// TIA Portal V19 export
FUNCTION_BLOCK "Area02_HU_FB"   // FB144, LAD
TITLE = AREA 01 HU PUMP
// stored: MemoryReserve 100, SetENOAutomatically false
   VAR_INPUT
      AreaInterface : "AreaInterface";
   END_VAR
   VAR_OUTPUT
      MachineInterface : "MachineInterface";
   END_VAR
   VAR
      Pump : "HU_Pump";
      Tank { S7_SetPoint := 'True'} : "HU_Tank";
      HMI : Struct
         Pressure_FinalCut : Real;
      END_STRUCT;
   END_VAR
   VAR_TEMP
      retval : Int;
      OilTemperature : Real;
      AnalTemperature_Real : Real;
      Delta : Real;
      Delta2 : Real;
   END_VAR
BEGIN

REGION Network 1: <<< PUMP >>>
END_REGION

REGION Network 2: Data In
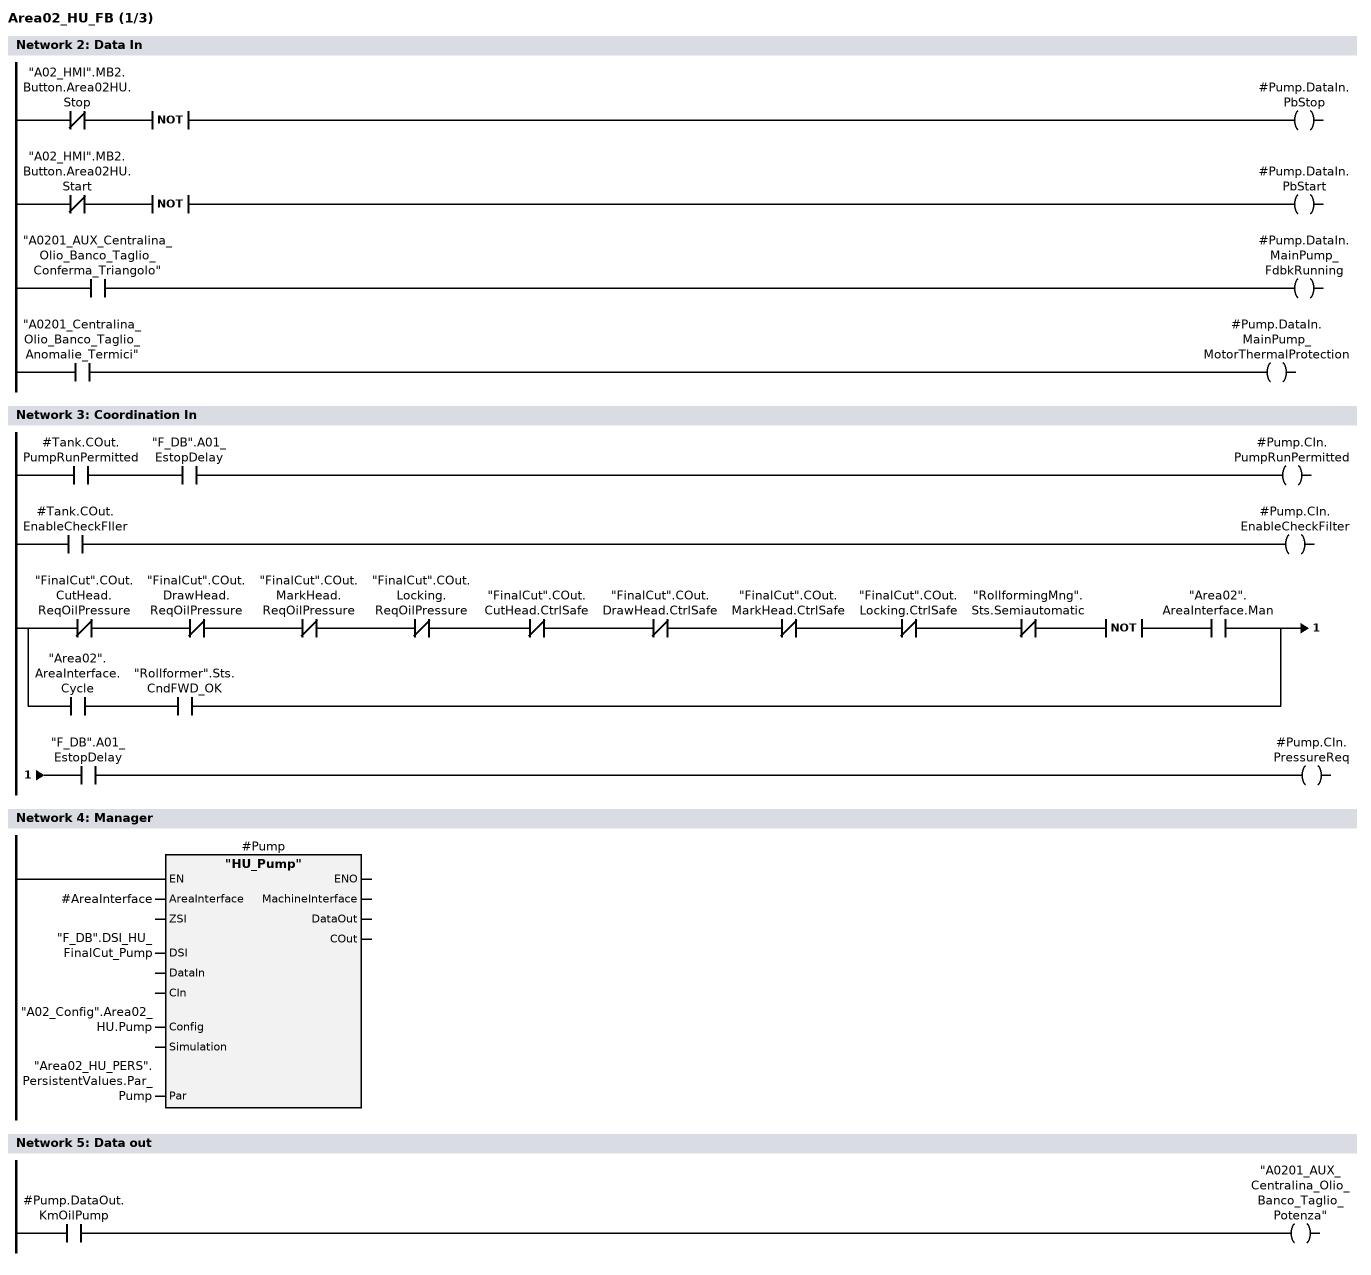
   RUNG wire#powerrail
      I_Contact( "A02_HMI".MB2.Button.Area02HU.Stop )
      Not()
      Coil( #Pump.DataIn.PbStop )
   END_RUNG
   RUNG wire#powerrail
      I_Contact( "A02_HMI".MB2.Button.Area02HU.Start )
      Not()
      Coil( #Pump.DataIn.PbStart )
   END_RUNG
   RUNG wire#powerrail
      Contact( "A0201_AUX_Centralina_Olio_Banco_Taglio_Conferma_Triangolo" )
      Coil( #Pump.DataIn.MainPump_FdbkRunning )
   END_RUNG
   RUNG wire#powerrail
      Contact( "A0201_Centralina_Olio_Banco_Taglio_Anomalie_Termici" )
      Coil( #Pump.DataIn.MainPump_MotorThermalProtection )
   END_RUNG
   // the same network as SCL:
   #Pump.DataIn.PbStop := NOT (NOT "A02_HMI".MB2.Button.Area02HU.Stop);
   #Pump.DataIn.PbStart := NOT (NOT "A02_HMI".MB2.Button.Area02HU.Start);
   #Pump.DataIn.MainPump_FdbkRunning := "A0201_AUX_Centralina_Olio_Banco_Taglio_Conferma_Triangolo";
   #Pump.DataIn.MainPump_MotorThermalProtection := "A0201_Centralina_Olio_Banco_Taglio_Anomalie_Termici";
END_REGION

REGION Network 3: Coordination In
   RUNG wire#powerrail
      Contact( #Tank.COut.PumpRunPermitted )
      Contact( "F_DB".A01_EstopDelay )
      Coil( #Pump.CIn.PumpRunPermitted )
   END_RUNG
   RUNG wire#powerrail
      Contact( #Tank.COut.EnableCheckFIler )
      Coil( #Pump.CIn.EnableCheckFilter )
   END_RUNG
   RUNG wire#powerrail
      I_Contact( "FinalCut".COut.CutHead.ReqOilPressure )
      I_Contact( "FinalCut".COut.DrawHead.ReqOilPressure )
      I_Contact( "FinalCut".COut.MarkHead.ReqOilPressure )
      I_Contact( "FinalCut".COut.Locking.ReqOilPressure )
      I_Contact( "FinalCut".COut.CutHead.CtrlSafe )
      I_Contact( "FinalCut".COut.DrawHead.CtrlSafe )
      I_Contact( "FinalCut".COut.MarkHead.CtrlSafe )
      I_Contact( "FinalCut".COut.Locking.CtrlSafe )
      I_Contact( "RollformingMng".Sts.Semiautomatic )
      Not()
      Contact( "Area02".AreaInterface.Man )
      wire#w1
      Contact( "F_DB".A01_EstopDelay )
      Coil( #Pump.CIn.PressureReq )
   END_RUNG
   RUNG wire#powerrail
      Contact( "Area02".AreaInterface.Cycle )
      Contact( "Rollformer".Sts.CndFWD_OK )
   END_RUNG wire#w1
   // the same network as SCL:
   #Pump.CIn.PumpRunPermitted := #Tank.COut.PumpRunPermitted AND "F_DB".A01_EstopDelay;
   #Pump.CIn.EnableCheckFilter := #Tank.COut.EnableCheckFIler;
   #Pump.CIn.PressureReq := ((NOT (NOT "FinalCut".COut.CutHead.ReqOilPressure AND NOT "FinalCut".COut.DrawHead.ReqOilPressure AND NOT "FinalCut".COut.MarkHead.ReqOilPressure AND NOT "FinalCut".COut.Locking.ReqOilPressure AND NOT "FinalCut".COut.CutHead.CtrlSafe AND NOT "FinalCut".COut.DrawHead.CtrlSafe AND NOT "FinalCut".COut.MarkHead.CtrlSafe AND NOT "FinalCut".COut.Locking.CtrlSafe AND NOT "RollformingMng".Sts.Semiautomatic) AND "Area02".AreaInterface.Man) OR ("Area02".AreaInterface.Cycle AND "Rollformer".Sts.CndFWD_OK)) AND "F_DB".A01_EstopDelay;
END_REGION

REGION Network 4: Manager
   RUNG wire#powerrail
      #Pump(AreaInterface := #AreaInterface, ZSI :=, DSI := "F_DB".DSI_HU_FinalCut_Pump, DataIn :=, CIn :=, Config := "A02_Config".Area02_HU.Pump, Simulation :=, Par := "Area02_HU_PERS".PersistentValues.Par_Pump, MachineInterface =>, DataOut =>, COut =>)
   END_RUNG
   // the same network as SCL:
   #Pump(AreaInterface := #AreaInterface,   // "HU_Pump"
         DSI := "F_DB".DSI_HU_FinalCut_Pump,
         Config := "A02_Config".Area02_HU.Pump,
         Par := "Area02_HU_PERS".PersistentValues.Par_Pump);
END_REGION

REGION Network 5: Data out
   RUNG wire#powerrail
      Contact( #Pump.DataOut.KmOilPump )
      Coil( "A0201_AUX_Centralina_Olio_Banco_Taglio_Potenza" )
   END_RUNG
   // the same network as SCL:
   "A0201_AUX_Centralina_Olio_Banco_Taglio_Potenza" := #Pump.DataOut.KmOilPump;
END_REGION

REGION Network 6: >
END_REGION

REGION Network 7: >
END_REGION

REGION Network 8: >
END_REGION

REGION Network 9: <<< TANK >>>
END_REGION

REGION Network 10: Data In
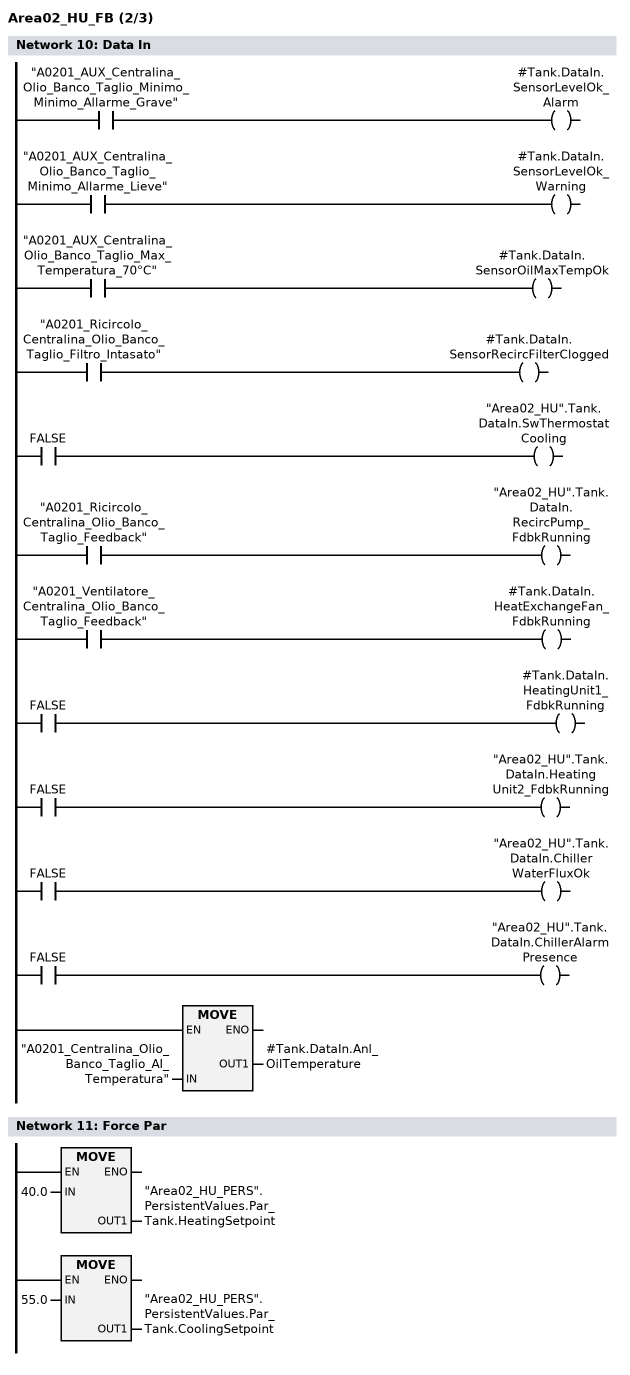
   RUNG wire#powerrail
      Contact( "A0201_AUX_Centralina_Olio_Banco_Taglio_Minimo_Minimo_Allarme_Grave" )
      Coil( #Tank.DataIn.SensorLevelOk_Alarm )
   END_RUNG
   RUNG wire#powerrail
      Contact( "A0201_AUX_Centralina_Olio_Banco_Taglio_Minimo_Allarme_Lieve" )
      Coil( #Tank.DataIn.SensorLevelOk_Warning )
   END_RUNG
   RUNG wire#powerrail
      Contact( "A0201_AUX_Centralina_Olio_Banco_Taglio_Max_Temperatura_70°C" )
      Coil( #Tank.DataIn.SensorOilMaxTempOk )
   END_RUNG
   RUNG wire#powerrail
      Contact( "A0201_Ricircolo_Centralina_Olio_Banco_Taglio_Filtro_Intasato" )
      Coil( #Tank.DataIn.SensorRecircFilterClogged )
   END_RUNG
   RUNG wire#powerrail
      Contact( FALSE )
      Coil( "Area02_HU".Tank.DataIn.SwThermostatCooling )
   END_RUNG
   RUNG wire#powerrail
      Contact( "A0201_Ricircolo_Centralina_Olio_Banco_Taglio_Feedback" )
      Coil( "Area02_HU".Tank.DataIn.RecircPump_FdbkRunning )
   END_RUNG
   RUNG wire#powerrail
      Contact( "A0201_Ventilatore_Centralina_Olio_Banco_Taglio_Feedback" )
      Coil( #Tank.DataIn.HeatExchangeFan_FdbkRunning )
   END_RUNG
   RUNG wire#powerrail
      Contact( FALSE )
      Coil( #Tank.DataIn.HeatingUnit1_FdbkRunning )
   END_RUNG
   RUNG wire#powerrail
      Contact( FALSE )
      Coil( "Area02_HU".Tank.DataIn.HeatingUnit2_FdbkRunning )
   END_RUNG
   RUNG wire#powerrail
      Contact( FALSE )
      Coil( "Area02_HU".Tank.DataIn.ChillerWaterFluxOk )
   END_RUNG
   RUNG wire#powerrail
      Contact( FALSE )
      Coil( "Area02_HU".Tank.DataIn.ChillerAlarmPresence )
   END_RUNG
   RUNG wire#powerrail
      { S7_GenerateENO := "TRUE" } Move(in := "A0201_Centralina_Olio_Banco_Taglio_AI_Temperatura", out1 => #Tank.DataIn.Anl_OilTemperature)
   END_RUNG
   // the same network as SCL:
   #Tank.DataIn.SensorLevelOk_Alarm := "A0201_AUX_Centralina_Olio_Banco_Taglio_Minimo_Minimo_Allarme_Grave";
   #Tank.DataIn.SensorLevelOk_Warning := "A0201_AUX_Centralina_Olio_Banco_Taglio_Minimo_Allarme_Lieve";
   #Tank.DataIn.SensorOilMaxTempOk := "A0201_AUX_Centralina_Olio_Banco_Taglio_Max_Temperatura_70°C";
   #Tank.DataIn.SensorRecircFilterClogged := "A0201_Ricircolo_Centralina_Olio_Banco_Taglio_Filtro_Intasato";
   "Area02_HU".Tank.DataIn.SwThermostatCooling := FALSE;
   "Area02_HU".Tank.DataIn.RecircPump_FdbkRunning := "A0201_Ricircolo_Centralina_Olio_Banco_Taglio_Feedback";
   #Tank.DataIn.HeatExchangeFan_FdbkRunning := "A0201_Ventilatore_Centralina_Olio_Banco_Taglio_Feedback";
   #Tank.DataIn.HeatingUnit1_FdbkRunning := FALSE;
   "Area02_HU".Tank.DataIn.HeatingUnit2_FdbkRunning := FALSE;
   "Area02_HU".Tank.DataIn.ChillerWaterFluxOk := FALSE;
   "Area02_HU".Tank.DataIn.ChillerAlarmPresence := FALSE;
   #Tank.DataIn.Anl_OilTemperature := "A0201_Centralina_Olio_Banco_Taglio_AI_Temperatura";
END_REGION

REGION Network 11: Force Par
   RUNG wire#powerrail
      { S7_GenerateENO := "TRUE" } Move(in := 40.0, out1 => "Area02_HU_PERS".PersistentValues.Par_Tank.HeatingSetpoint)
   END_RUNG
   RUNG wire#powerrail
      { S7_GenerateENO := "TRUE" } Move(in := 55.0, out1 => "Area02_HU_PERS".PersistentValues.Par_Tank.CoolingSetpoint)
   END_RUNG
   // the same network as SCL:
   "Area02_HU_PERS".PersistentValues.Par_Tank.HeatingSetpoint := 40.0;
   "Area02_HU_PERS".PersistentValues.Par_Tank.CoolingSetpoint := 55.0;
END_REGION

REGION Network 12: HMI Pressure
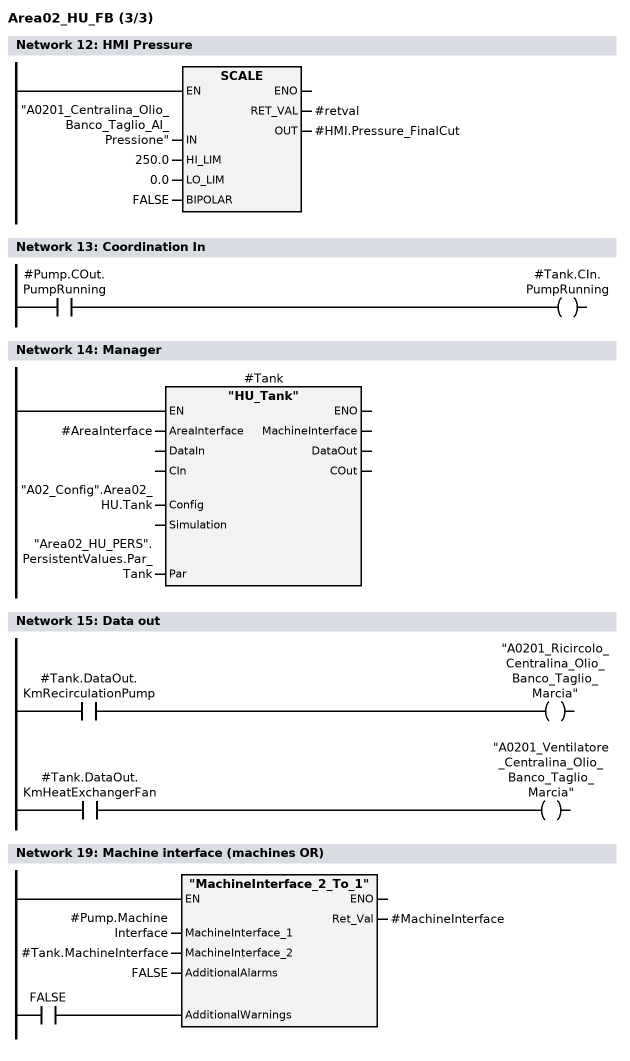
   #retval := SCALE(IN := "A0201_Centralina_Olio_Banco_Taglio_AI_Pressione",
                    HI_LIM := 250.0,
                    LO_LIM := 0.0,
                    BIPOLAR := FALSE,
                    OUT => #HMI.Pressure_FinalCut);
END_REGION

REGION Network 13: Coordination In
   RUNG wire#powerrail
      Contact( #Pump.COut.PumpRunning )
      Coil( #Tank.CIn.PumpRunning )
   END_RUNG
   // the same network as SCL:
   #Tank.CIn.PumpRunning := #Pump.COut.PumpRunning;
END_REGION

REGION Network 14: Manager
   RUNG wire#powerrail
      #Tank(AreaInterface := #AreaInterface, DataIn :=, CIn :=, Config := "A02_Config".Area02_HU.Tank, Simulation :=, Par := "Area02_HU_PERS".PersistentValues.Par_Tank, MachineInterface =>, DataOut =>, COut =>)
   END_RUNG
   // the same network as SCL:
   #Tank(AreaInterface := #AreaInterface,   // "HU_Tank"
         Config := "A02_Config".Area02_HU.Tank,
         Par := "Area02_HU_PERS".PersistentValues.Par_Tank);
END_REGION

REGION Network 15: Data out
   RUNG wire#powerrail
      Contact( #Tank.DataOut.KmRecirculationPump )
      Coil( "A0201_Ricircolo_Centralina_Olio_Banco_Taglio_Marcia" )
   END_RUNG
   RUNG wire#powerrail
      Contact( #Tank.DataOut.KmHeatExchangerFan )
      Coil( "A0201_Ventilatore_Centralina_Olio_Banco_Taglio_Marcia" )
   END_RUNG
   // the same network as SCL:
   "A0201_Ricircolo_Centralina_Olio_Banco_Taglio_Marcia" := #Tank.DataOut.KmRecirculationPump;
   "A0201_Ventilatore_Centralina_Olio_Banco_Taglio_Marcia" := #Tank.DataOut.KmHeatExchangerFan;
END_REGION

REGION Network 16: >
END_REGION

REGION Network 17: >
END_REGION

REGION Network 18: >
END_REGION

REGION Network 19: Machine interface (machines OR)
   RUNG wire#powerrail
      "MachineInterface_2_To_1"(AdditionalWarnings := wire#w1, MachineInterface_1 := #Pump.MachineInterface, MachineInterface_2 := #Tank.MachineInterface, AdditionalAlarms := FALSE, Ret_Val => #MachineInterface)
   END_RUNG
   RUNG wire#powerrail
      Contact( FALSE )
   END_RUNG wire#w1
   // the same network as SCL:
   #MachineInterface := "MachineInterface_2_To_1"(MachineInterface_1 := #Pump.MachineInterface,
                           MachineInterface_2 := #Tank.MachineInterface,
                           AdditionalAlarms := FALSE,
                           AdditionalWarnings := FALSE);
END_REGION
END_FUNCTION_BLOCK
